INTERFACE I_InputPortChangedEvent EXTENDS I_Event

PROPERTY PUBLIC Target : I_InputPort
GET
END_GET
END_PROPERTY

END_INTERFACE

(* stored: Version 1.1.0.1, ProductVersion 3.1.4024.12
   Itf I_InputPortChangedEvent: Id {3c66a25d-98eb-482e-8bb1-f1bdba844aa2}
   Property Target: Id {cdb9b483-b318-4a2d-ba1a-04509af97b7b}
   Get Get: Id {ff2e36ce-d289-418d-a5c6-2b14433979a5} *)
